TYPE Vec2i : ARRAY[1..2] OF INT; END_TYPE

(* stored: Version 1.1.0.1, ProductVersion 3.1.4024.11
   DUT Vec2i: Id {4d9fe461-8cca-48f1-a1f7-47974c47d723} *)
